(* CODESYS project RFID_Sorter_SP11.project

Project tree, tasks and I/O mapping:
  Device : TBEN-Lx-PLC-1x, Turck, version 3.5.16.20
    application Application
      libraries: Standard, 3.5.18.0 (System); BASIC, 3.3.4.0 (OSCAT); Util, 3.5.19.0 (System)
      task MainTask (cyclic, interval 20 ms, priority 1) calls PLC_PRG
      program PLC_PRG [ST]: ACT_READ_REGISTERS, ACT_SET_REGISTERS, MODBUS
      function FUN_CONVEYOR_SELECTOR [ST]
    LEDs : LEDs, Turck, version 1.1.1.0
        unmapped channels: LED 4 (green), LED 4 (red), LED 5 (green), LED 5 (red), LED 6 (green), LED 6 (red), LED 7 (green), LED 7 (red), APPL LED (green), APPL LED (red)
    Local_IO : Local IO, Turck, version 1.0.2.0
      DXP : DXP, Turck, version 1.0.2.0
          unmapped channels: DXP, DXP
      Diagnostics : Diagnostics, Turck, version 1.0.2.0
          unmapped channels: Diagnostics
      VAUX_control : VAUX control, Turck, version 1.0.2.0
          unmapped channels: VAUX control
      Module_status : Module status, Turck, version 1.0.2.0
          unmapped channels: Module status
    COM0
    COM1
    CANbus
    Ethernet : Ethernet, Turck, version 3.5.16.20
        settings: IPAddress = [10,6,2,211]; SubnetMask = [255,255,252,0]; GatewayAddress = [10,6,0,1]; MACAddress = [16#00,16#07,16#46,16#8D,16#62,16#F3]; SaveCommunicationSettings = FALSE
      Modbus_TCP_Master : Modbus TCP Master, 3S - Smart Software Solutions GmbH, version 3.5.14.0
        Modbus_TCP_Slave : Modbus TCP Slave, 3S - Smart Software Solutions GmbH, version 4.1.0.0
            settings: Unit-ID = 255; IPAddress = [10, 6, 2, 200]
*)

// Device/Application/PLC_PRG
PROGRAM PLC_PRG
VAR
	READ_TIMEOUT : TIME;
	MODBUS_SLAVE_READ : IoDrvModbusTCP.ModbusRequest;
	xExecute : BOOL;
	xAbort : BOOL;
	xDone : BOOL;
	xBusy : BOOL;
	xError : BOOL;
	xAborted : BOOL;
	Modbus_Command : IoDrvModbusTCP.ModbusCommand;
	usiUnitID : USINT := 1;
	ModbusError : IoDrvModbusTCP.MB_ErrorCodes;
	abySendData : ARRAY[0..127] OF WORD;
	abyRecvData : ARRAY[0..127] OF WORD;
	udiUpdateCommSettings : UDINT;
	
	// conveyor variables
	// sensors
	xDiffuseSensorSource : BOOL;
	xDiffuseSensorSource0 : BOOL;
	xDiffuseSensorRight : BOOL;
	xDiffuseSensorFeeder : BOOL;
	//conveyors
	xRollerConveyorSource : BOOL;
	xRollerConveyorSource0 : BOOL;
	xRollerConveyorLeft : BOOL;
	xRollerConveyorRight : BOOL;
	xRollerConveyorStraight : BOOL;
	//turn table
	xTurnTableRollFront : BOOL;
	xTurnTableRollBack : BOOL;
	xTurnTableTurn : BOOL;
	xTurnTableLimit0 : BOOL;
	xTurnTableLimit90 : BOOL;
	xTurnTableLimitFront : BOOL;
	xTurnTableLimitBack : BOOL;
	
	
	iRunConveyor : INT := 1;
	xStart : BOOL;
	xReset : BOOL;
	xRunning : BOOL;
	
	xRunConveyor : BOOL;
	xResetConveyor : BOOL;
	xPauseConveyor : BOOL;
	wWordConvert: Util.WORD_AS_BIT;
	
	
	iReadData : INT := 1;
	xReadData : BOOL;
	iSendData : INT := 1;;
	xSendData : BOOL;
	
	iPalletCounter : INT;
	iFeederConveyor : INT := 1;
	xPalletOnConveyor : BOOL;
	xFeederTagDetected : BOOL;
	xFeederTagCommand : BOOL;
	xFeederTagcommandExecute : BOOL;
	
	// modbus
	iModbusComm : INT := 1;
	
	// RFID feeder
	ifRFID_Command : INT;
	ifRFID_CommandID : INT;
	ifRFID_PrevCommandID : INT;
	ifRFID_Status : INT;
	ifRFID_WriteData : INT;
	xfRFID_CommandExecute : BOOL;
	
	// RFID main conveyor
	imRFID_Command : INT;
	imRFID_CommandID : INT;
	imRFID_PrevCommandID : INT;
	imRFID_Status : INT;
	imRFID_ReadData : INT;
	xmRFID_CommandExecute : BOOL;
	
	// emitter
	xFeederEmitterEmit : BOOL;
	iCount : INT;
	
	tDelay : TON;
	tDelay2 : TON;
	
	// TAGS
	iEpctag : INT;
	iSelectedConveyor : INT;
	
	xLeftConveyorSelected : BOOL;
	iLeftConveyorRun : INT := 1;
	xStraightConveyorSelected : BOOL;
	iStraightConveyorRun : INT := 1;
	xRightConveyorSelected : BOOL;
	iRightConveyorRun : INT := 1;
	
	
	
	
END_VAR

Modbus_Command.uiReadOffset := 0;
Modbus_Command.uiWriteOffset := 0;
usiUnitID := 1;	

// time delay for Feeder conveyor RFID Reader 
tDelay(IN:= , PT:=T#4S, Q=>);
// Time delay for Main conveyor RFID Reader
tDelay2(IN:= , PT:=T#4S, Q=>);

// modbus comm 
CASE iModbusComm OF
	1:
	IF xStart OR xReset THEN
		xSendData := TRUE;
		iModbusComm := 2;
	END_IF
	
	2:
	IF NOT xSendData THEN
		IF xReset THEN
			xReset := FALSE;
		END_IF
		xReadData := TRUE;
		iModbusComm := 3;
	END_IF
	
	3:
	IF NOT xReadData THEN
		iModbusComm := 1;
	END_IF
END_CASE
	
// Send Data to modbus server
ACT_READ_REGISTERS();
// Read data from Modbus Server
ACT_SET_REGISTERS();
// Run Modbus Reguest block
MODBUS();

// feeder conveyor 0
CASE iFeederConveyor OF
	1:
	// emit pallet if there id no pallet on main conveyor
	IF xStart AND NOT xPalletOnConveyor THEN
		xRollerConveyorSource0 := TRUE;
		xFeederEmitterEmit := TRUE;
		ifRFID_PrevCommandID := ifRFID_CommandID;
		iEpctag := iEpctag +1;
		iFeederConveyor := 2;
	END_IF
	
	2:
	// stop conveyor when packet is detected by feeder sensor
	IF xDiffuseSensorFeeder THEN
		xFeederEmitterEmit := FALSE;
		xRollerConveyorSource0 := FALSE;
		iFeederConveyor := 3;
	END_IF
	
	3:
	// write new epc to package tag
	IF (tDelay.IN  AND tDelay.Q) OR NOT tDelay.IN THEN
		tDelay.IN := FALSE;
		ifRFID_WriteData := iEpctag;
		ifRFID_Command := 3;
		xfRFID_CommandExecute := TRUE;
		iFeederConveyor := 4;
	END_IF
	
	4:
	// if write operation is not successful, try again
	IF ifRFID_PrevCommandID <> ifRFID_CommandID THEN
		IF ifRFID_Status = 0 THEN
			xfRFID_CommandExecute := FALSE;
			iFeederConveyor := 5;
		ELSE
			tDelay.IN := TRUE;
			xfRFID_CommandExecute := FALSE;
			ifRFID_PrevCommandID := ifRFID_CommandID;
			iFeederConveyor := 3;
		END_IF
	END_IF
	
	5:
	// restart feeder conveyor
	xRollerConveyorSource0 := TRUE;
	iFeederConveyor := 6;
	
	6:
	// stop feeder conveyor when packet arrives on main conveyor
	IF xPalletOnConveyor THEN
		xRollerConveyorSource0 := FALSE;
		iFeederConveyor := 1;
	END_IF
	
END_CASE

// main conveyor
CASE iRunConveyor OF 
	1: 
	// if system already running 
	IF xStart AND xRunning THEN
		// start main conveyor
		xRollerConveyorSource := TRUE;
		// update pallet counter
		iPalletCounter := iPalletCounter + 1;
		iRunConveyor := 2;
	// system start
	ELSIF xStart THEN
		// set state to running
		xRunning := TRUE; 
		// update pallet counter
		iPalletCounter := iPalletCounter + 1;
		// start application and reset all values
		xRunConveyor := TRUE;
		xResetConveyor := TRUE;
		// start main conveyor and destination conveyors
		xRollerConveyorSource := TRUE;
		xRollerConveyorLeft:= TRUE;
		xRollerConveyorRight := TRUE;
		xRollerConveyorStraight := TRUE;
		iRunConveyor := 2;
	END_IF
	
	2:
	// if pallet is detected by main conveyor sensor0, then pallet on conveyor
	IF xDiffuseSensorSource0 = TRUE THEN
		xPalletOnConveyor := TRUE;
		iRunConveyor := 3;
	END_IF	
	
	3:
	// if pallet is detected by main conveyor sensor1, stop conveyor and alight turn table
	IF xDiffuseSensorSource = TRUE THEN
		xRollerConveyorSource := FALSE;
		IF xTurnTableLimit0 THEN
			xTurnTableTurn := TRUE;
		END_IF
		imRFID_PrevCommandID := imRFID_CommandID;
		iRunConveyor := 10;
	END_IF	
	
	10:
	// read rfid tag
	IF (tDelay2.IN  AND tDelay2.Q) OR NOT tDelay2.IN THEN
		tDelay2.IN := FALSE;
		imRFID_Command := 2;
		xmRFID_CommandExecute := TRUE;
		iRunConveyor := 11;
	END_IF
	
	11:
	// if reading is not successfull, try again
	IF imRFID_PrevCommandID <> imRFID_CommandID THEN
		IF imRFID_Status = 0 THEN
			xmRFID_CommandExecute := FALSE;
			iRunConveyor := 4;
		ELSE
			xmRFID_CommandExecute := FALSE;
			tDelay2.IN := TRUE;
			imRFID_PrevCommandID := imRFID_CommandID;
			iRunConveyor := 10;
		END_IF
	END_IF
	
	4:
	// analyse read tag value and select destination conveyor
	iSelectedConveyor := FUN_CONVEYOR_SELECTOR(imRFID_ReadData);
	IF iSelectedConveyor = 1 THEN
		xLeftConveyorSelected := TRUE;
		iRunConveyor := 5;
	ELSIF iSelectedConveyor = 2 THEN
		xStraightConveyorSelected := TRUE;
		iRunConveyor := 5;
	ELSIF iSelectedConveyor = 3 THEN
		xRightConveyorSelected := TRUE;
		iRunConveyor := 5;
	END_IF
	
	5:
	// if pallet is delivered to destination conveyor, reset turn table and start again to handle next apllet
	IF NOT xLeftConveyorSelected AND NOT xStraightConveyorSelected AND NOT xRightConveyorSelected THEN
		xTurnTableRollBack := FALSE;
		xTurnTableRollFront := FALSE;
		iRunConveyor := 1;
	END_IF

END_CASE


// LEFT CONVEYOR
CASE iLeftConveyorRun OF 
	1:
	// if left conveor is selected
	IF xLeftConveyorSelected THEN
		iLeftConveyorRun := 2;
	END_IF
	
	2:
	// check if turn table is aligned then roll pallet on turn table
	IF xTurnTableLimit90 THEN
		xRollerConveyorSource := TRUE;
		xTurnTableRollBack := TRUE;
		iLeftConveyorRun := 3;
	END_IF
	
	3:
	// if pallet reaches end of turn table, then stop rolling, align turn table with left conveyor
	IF xTurnTableLimitBack THEN 
		xRollerConveyorSource := FALSE;
		xTurnTableRollBack := FALSE;
		xTurnTableTurn := FALSE;  //turn back
		iLeftConveyorRun := 4;
	END_IF
	
	4:
	// if aligned, push pallet to left conveyor, notify that pallent no longer on main conveyor
	IF xTurnTableLimit0 THEN
		xPalletOnConveyor := FALSE;
		xTurnTableRollFront := TRUE;
		iLeftConveyorRun := 5;
	END_IF
	
	5:
	IF xTurnTableLimitFront THEN
		iLeftConveyorRun := 6;
	END_IF
	
	6:
	// if pallet has cleared the turn table, give back control to main conveyor
	IF NOT xTurnTableLimitFront THEN
		xLeftConveyorSelected := FALSE;
		iLeftConveyorRun := 1;
	END_IF
	
END_CASE


// STRAIGHT CONVEYOR
CASE iStraightConveyorRun OF 
	1:
	// if straight conveor is selected
	IF xStraightConveyorSelected THEN
		iStraightConveyorRun := 2;
	END_IF
	
	2:
	// check if turn table is aligned then roll pallet on turn table
	IF xTurnTableLimit90 THEN
		xRollerConveyorSource := TRUE;
		xTurnTableRollBack := TRUE;
		iStraightConveyorRun := 3;
	END_IF
	
	3:
	// continue rolling until pallet clears turn table
	IF xTurnTableLimitBack THEN 
		xRollerConveyorSource := FALSE;
		xPalletOnConveyor := FALSE;
		iStraightConveyorRun := 4;
	END_IF
	
	4:
	iStraightConveyorRun := 5;
	
	5:
	// if pallet has cleared the turn table, give back control to main conveyor
	IF NOT xTurnTableLimitBack THEN
		xStraightConveyorSelected := FALSE;
		iStraightConveyorRun := 1;
	END_IF
	
END_CASE

// RIGHT CONVEYOR
CASE iRightConveyorRun OF 
	1:
	// if right conveor is selected
	IF xRightConveyorSelected THEN
		iRightConveyorRun := 2;
	END_IF
	
	2:
	// check if turn table is aligned then roll pallet on turn table
	IF xTurnTableLimit90 THEN
		xRollerConveyorSource := TRUE;
		xTurnTableRollBack := TRUE;
		iRightConveyorRun := 3;
	END_IF
	
	3:
	// if pallet reaches end of turn table, then stop rolling, align turn table with left conveyor
	IF xTurnTableLimitBack THEN 
		xRollerConveyorSource := FALSE;
		xTurnTableRollBack := FALSE;
		xTurnTableTurn := FALSE; 
		iRightConveyorRun := 4;
	END_IF
	
	4:
	// if aligned, push pallet to right conveyor, notify that pallent no longer on main conveyor
	IF xTurnTableLimit0 THEN
		xPalletOnConveyor := FALSE;
		xTurnTableRollBack := TRUE;
		xRollerConveyorRight := TRUE;
		iRightConveyorRun := 5;
	END_IF
	
	5:
	//if pallet clears turn table, give back control to main conveyor
	IF NOT xTurnTableLimitBack THEN
		xRightConveyorSelected := FALSE;
		iRightConveyorRun := 1;
	END_IF
	
END_CASE


	

// reset all parameters to initial values
IF xReset THEN
	xRollerConveyorSource0 := FALSE;
	xRollerConveyorSource:= FALSE;
	xRollerConveyorLeft:= FALSE;
	xRollerConveyorRight:= FALSE;
	xRollerConveyorStraight:= FALSE;
		//turn table
	xTurnTableTurn:= FALSE;
	xTurnTableRollFront:= FALSE;
	xTurnTableRollBack:= FALSE;
	xRunConveyor := TRUE;
	xResetConveyor := FALSE;
	
	xfRFID_CommandExecute := FALSE;
	ifRFID_CommandID := 0;
	xRunning := FALSE;
	iPalletCounter := 0;
	xStart := FALSE;	

	xPalletOnConveyor := FALSE;
	iFeederConveyor := 1;
	iRunConveyor := 1;
	
	iPalletCounter := 0;
	iFeederConveyor := 1;
	xPalletOnConveyor := FALSE;
	xFeederTagDetected := FALSE;
	xFeederTagCommand := FALSE;
	xFeederTagcommandExecute := FALSE;
	
		// RFID feeder
	ifRFID_Command := 0;
	ifRFID_CommandID := 0;
	ifRFID_PrevCommandID := 0;
	ifRFID_Status := 0;
	ifRFID_WriteData := 0;
	xfRFID_CommandExecute := FALSE;
	
		// RFID main conveyor
	imRFID_Command := 0;
	imRFID_CommandID := 0;
	imRFID_PrevCommandID := 0;
	imRFID_Status := 0;
	imRFID_ReadData := 0;
	xmRFID_CommandExecute := FALSE;
	
	iSelectedConveyor := 0;
	
	xLeftConveyorSelected := FALSE;
	iLeftConveyorRun := 1;
	xStraightConveyorSelected := FALSE;
	iStraightConveyorRun := 1;
	xRightConveyorSelected := FALSE;
	iRightConveyorRun := 1;
	
END_IF

ACTION ACT_READ_REGISTERS:

CASE iReadData OF
	1:
	// reads discrete inputs
	IF xReadData THEN
		Modbus_Command.FunctionCode := 2;
		Modbus_Command.uiReadLen := 16;
		xExecute := TRUE;
		iReadData := 2;
	END_IF
	2:
	// updates parameter values
	IF xDone THEN
		xDiffuseSensorSource := abyRecvData[0].0;
		xDiffuseSensorSource0 := abyRecvData[0].1;
		xDiffuseSensorRight := abyRecvData[0].2;
		xTurnTableLimit0 := abyRecvData[0].3;
		xTurnTableLimit90 := abyRecvData[0].4;
		xTurnTableLimitBack  := abyRecvData[0].5;
		xTurnTableLimitFront := abyRecvData[0].6;
		xDiffuseSensorFeeder := abyRecvData[0].7;
		xExecute := FALSE;
		iReadData := 3;
	END_IF
	
	3:
	// reads input registers
	IF NOT xDone THEN
		Modbus_Command.FunctionCode := 4;
		Modbus_Command.uiReadLen := 8;
		xExecute := TRUE;
		iReadData := 4;		
	END_IF
	
	4:
	// updates paramters
	IF xDone THEN
		ifRFID_Status := WORD_TO_INT(abyRecvData[4]);
		ifRFID_CommandID := WORD_TO_INT(abyRecvData[5]);
		
		imRFID_Status := WORD_TO_INT(abyRecvData[0]);
		imRFID_ReadData := WORD_TO_INT(abyRecvData[1]);
		imRFID_CommandID := WORD_TO_INT(abyRecvData[2]);
		xExecute := FALSE;
		xReadData := FALSE;
		iReadData := 1;
	END_IF
END_CASE
END_ACTION

ACTION ACT_SET_REGISTERS:

CASE iSendData OF
	1:
	// updates registers and sets coils
	IF xSendData THEN
		abySendData[0].0 := xRollerConveyorSource0;
		abySendData[0].1 := xRollerConveyorSource;
		abySendData[0].2 := xRollerConveyorLeft;
		abySendData[0].3 := xRollerConveyorRight;
		abySendData[0].4 := xRollerConveyorStraight;
		//turn table
		abySendData[0].5 := xTurnTableTurn;
		abySendData[0].6 := xTurnTableRollFront;
		abySendData[0].7 := xTurnTableRollBack;
		abySendData[0].8 := xmRFID_CommandExecute;
		abySendData[0].9 := xfRFID_CommandExecute ;
		
		
		abySendData[0].10 :=	xRunConveyor;
		abySendData[0].11 :=	xResetConveyor;
		abySendData[0].12 :=	xPauseConveyor ;
		
		// EMITTER
		abySendData[0].15 := xFeederEmitterEmit;	
		
		Modbus_Command.FunctionCode := 15;
		Modbus_Command.uiWriteLen := 16;
		
		xExecute := TRUE;
		iSendData := 2;
	END_IF
	
	2:
	IF xDone THEN
		xExecute := FALSE;
		iSendData := 3;
	END_IF
	
	3:
	//updates registers and sets holding registers
	IF NOT xDone THEN
		abySendData[0] := 0;
		abySendData[4] := INT_TO_WORD(ifRFID_Command) ;
		abySendData[5] := INT_TO_WORD(ifRFID_WriteData);
		abySendData[6] := INT_TO_WORD(imRFID_Command);
		
		Modbus_Command.FunctionCode := 16;
		Modbus_Command.uiWriteLen := 8;
		xExecute := TRUE;
		iSendData := 4;
	END_IF
	
	4:
	IF xDone THEN
		xExecute := FALSE;
		xSendData := FALSE;
		iSendData := 1;
	END_IF
END_CASE
END_ACTION

ACTION MODBUS:
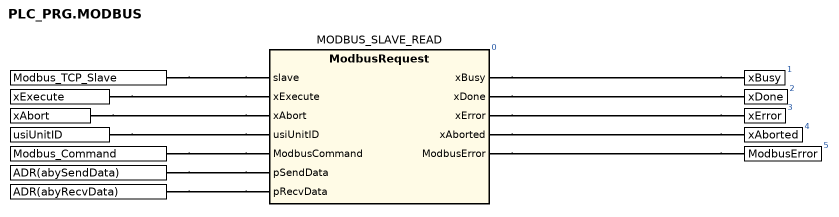
MODBUS_SLAVE_READ(
    slave := Modbus_TCP_Slave,
    xExecute := xExecute,
    xAbort := xAbort,
    usiUnitID := usiUnitID,
    ModbusCommand := Modbus_Command,
    pSendData := ADR(abySendData),
    pRecvData := ADR(abyRecvData)); // ModbusRequest
xBusy := MODBUS_SLAVE_READ.xBusy;
xDone := MODBUS_SLAVE_READ.xDone;
xError := MODBUS_SLAVE_READ.xError;
xAborted := MODBUS_SLAVE_READ.xAborted;
ModbusError := MODBUS_SLAVE_READ.ModbusError;
END_ACTION

END_PROGRAM

// Device/Application/FUN_CONVEYOR_SELECTOR
FUNCTION FUN_CONVEYOR_SELECTOR : INT
VAR_INPUT
	iTag : INT;
END_VAR
VAR
END_VAR

FUN_CONVEYOR_SELECTOR := 0;
IF iTag MOD 2 = 0 THEN
	IF iTag MOD 4 = 0 THEN
		FUN_CONVEYOR_SELECTOR := 3;
	ELSE
		FUN_CONVEYOR_SELECTOR := 2;
	END_IF
ELSE
	FUN_CONVEYOR_SELECTOR := 1;
END_IF

END_FUNCTION
